PROGRAM MAIN
VAR
	stGyroAxis AT %I* : ST_3d_values;
	stcorrAxis : ST_3d_values;
	stOffset	:ST_3d_values;

	fbMovingAverage_3D: FB_MovingAverageFilter_3D;
	a_fBuffer : ARRAY[0..2] OF ARRAY[ 0..GVL_SensorFusion.buffersize_filter-1] OF REAL;
	
(* Accelerometer values *)
	stAccAxis AT %I* : ST_3d_values;
	normalizedAcceleration : ARRAY [0..2] OF LREAL;

(* Working variables *)
	fbStartOffsetCalibration : R_TRIG;
	bReset: BOOL;
	fbOffsetSet : R_TRIG;
	bResetAngles: BOOL;

	fCycleTime 				: LREAL; // PLC cycle time in s (has to match with ODR of sensor => for prototype this is static 4000Hz)
	nTaskIndex				: DINT;
	bReady					: BOOL;
	
(*Disclaimer: This is a sample still in prototype phase.
Please be aware that functionalities/ PDOs / CoEs can differ in series variant.
*)
	fbKalmanFilter:FB_KalmanFilter;
	fbMadgwickFilter:FB_MadgwickFilter;
	fbComplementaryFilter:FB_ComplementaryFilter;
	fbMahonyFilter:FB_MahonyFilter;
	stEulerAngle_Gyro:ST_3D_Values;
END_VAR

nTaskIndex:=GETCURTASKINDEXEX();
IF nTaskIndex>0 THEN
	fCycletime:=UDINT_TO_LREAL(_TaskInfo[GETCURTASKINDEXEX()].CycleTime) / 10_000_000;
END_IF

// get Sensoroffset
fbStartOffsetCalibration(clk:=bReset);
	

fbMovingAverage_3D( stSampleData:=stGyroAxis, bEnable:=NOT fbStartOffsetCalibration.Q, a_fSamples:=a_fBuffer);
fbOffsetSet(clk:=fbMovingAverage_3D.bBufferFilledX);
IF fbOffsetSet.Q THEN
	stOffset.x:=fbMovingAverage_3D.stAvgData.X;
	stOffset.y:=fbMovingAverage_3D.stAvgData.y;
	stOffset.z:=fbMovingAverage_3D.stAvgData.z;
	stEulerAngle_Gyro.x:=0;
	stEulerAngle_Gyro.y:=0;
	stEulerAngle_Gyro.z:=0;
	bResetAngles:=TRUE;
ELSIF bResetAngles THEN
	stEulerAngle_Gyro.x:=0;
	stEulerAngle_Gyro.y:=0;
	stEulerAngle_Gyro.z:=0;
END_IF

bReady:=fbMovingAverage_3D.bBufferFilledX;

//correct Gyro-Values with Offset
stcorrAxis.X:= stGyroAxis.X - stOffset.x;
stcorrAxis.Y:= stGyroAxis.Y - stOffset.y;
stcorrAxis.Z:= stGyroAxis.Z - stOffset.z;


	//Calculate Euler Angles by Sensorfusion
	fbKalmanFilter(
		stAccelData:= stAccAxis, 
		stGyroData:= stcorrAxis,  
		fCycleTime:= fCycletime,
		bSetReference:=bResetAngles );
		
	fbMadgwickFilter(
		stAccelData:= stAccAxis, 
		stGyroData:= stcorrAxis,  
		fcycletime:=fCycletime , 
		bSetReference:= bResetAngles );
		
	fbComplementaryFilter(
		stAccelData:= stAccAxis, 
		stGyroData:= stcorrAxis,  
		fcycletime:=fCycletime , 
		bSetReference:= bResetAngles );
		
	fbMahonyFilter(
		stAccelData:= stAccAxis, 
		stGyroData:= stcorrAxis,  
		fcycletime:=fCycletime , 
		bSetReference:= bResetAngles );

bResetAngles:=FALSE;
stEulerAngle_Gyro.x := stEulerAngle_Gyro.x + stcorrAxis.x * fCycleTime;
stEulerAngle_Gyro.y := stEulerAngle_Gyro.y + stcorrAxis.y * fCycleTime;
stEulerAngle_Gyro.z := stEulerAngle_Gyro.z + stcorrAxis.Z * fCycleTime;

END_PROGRAM

(* stored: Version 1.1.0.1, ProductVersion 3.1.4024.15
   POU MAIN: Id {5ed6dd28-4e50-4912-a842-bd2821892fe5}, SpecialFunc None *)
